INTERFACE I_Mc3AxisRef

PROPERTY Axis : REFERENCE TO Tc3_Mc3Ptp.AXIS_REF
GET
END_GET
END_PROPERTY

END_INTERFACE

(* stored: Version 1.1.0.1, ProductVersion 3.1.4026.20
   Itf I_Mc3AxisRef: Id {cfa22f24-7e51-4c91-b465-c94480e085c3}
   Property Axis: Id {3b2e3525-5303-4a8c-8754-780624ae36ff}
   Get Get: Id {edf8c2c5-ddc4-42ed-a80a-1a48f11c4518} *)
